// Iteration helper method to iterate from a given node in a specific direction for a specified count.
METHOD PROTECTED Iterate : POINTER TO T_List_Node
VAR_INPUT
	pStart 		: POINTER TO T_List_Node;
	Count 		: T_Capacity;
	bIterateUp 	: BOOL;
END_VAR
VAR
	i : T_Capacity;
END_VAR
Iterate := pStart;
IF Count = 0 THEN RETURN; END_IF
IF bIterateUp THEN FOR i := 0 TO Count - 1 DO Iterate := Iterate^.pNext; END_FOR RETURN; END_IF
FOR i := 0 TO Count - 1 DO Iterate := Iterate^.pPrevious; END_FOR
END_METHOD

// Adds an item to the end of the list.
METHOD Append : I_List
VAR_INPUT
	Item : ANY; // Value to store in list
END_VAR
VAR_OUTPUT
	bSuccess : BOOL;
END_VAR
Append := THIS^;

THIS^.Insert_Generic(THIS^._Count, Item, bSuccess => bSuccess);
END_METHOD

// Empties/Clears/Deletes every item in the list.
METHOD Clear : I_List
VAR
	pTmp : POINTER TO T_List_Node;
END_VAR
Clear := THIS^;

WHILE THIS^.pHead <> 0 DO
	pTmp := THIS^.pHead^.pNext;
	F_Delete_Generic(THIS^.pHead^.Data);
	__DELETE(THIS^.pHead);
	THIS^.pHead := pTmp;
	END_WHILE

THIS^._Count := 0;	
THIS^.pTail := THIS^.pLast_Accessed := 0;
THIS^.Last_Accessed_Index := -1;
THIS^.Clear_Error();
END_METHOD

// Checks if item is contained in list.
METHOD Contains : BOOL
VAR_INPUT
	Item : ANY; // Item to find in list
END_VAR
THIS^.Search(Item, bSuccess => Contains);
END_METHOD

METHOD FB_exit : BOOL
VAR_INPUT
	bInCopyCode : BOOL; // if TRUE, the exit method is called for exiting an instance that is copied afterwards (online change).
END_VAR
THIS^.Clear();
END_METHOD

// Gets item from list at specified location without removing it
METHOD Get : I_List
VAR_INPUT
	Index : T_Position; // Location of item
	Item : ANY;  // Variable to store returned item
END_VAR
VAR_OUTPUT
	bSuccess : BOOL;
END_VAR
VAR
	Tmp : T_Generic;
END_VAR
Get := THIS^;

THIS^.Get_Generic(Index, Item => Tmp, bSuccess => bSuccess);

IF NOT bSuccess THEN RETURN; END_IF

IF NOT F_Matching_Generics(Item, Tmp) THEN
	THIS^._Error_Status := F_Error(TRUE, GVL_Errors.ERR_TYPE_MISMATCH, 'Type mismatch.');
	RETURN;
	END_IF
	
F_Copy_Generic_Value(Tmp, Item);
bSuccess := TRUE;
THIS^.Clear_Error();
END_METHOD

// Returns item as a string, if type to string conversion is supported
METHOD Get_As_String : I_List
VAR_INPUT
	Index : T_Position; // Location of item
	sItem : REFERENCE TO STRING; // Variable to store returned item.
END_VAR
VAR_OUTPUT
	bSuccess : BOOL;
END_VAR
VAR
	Tmp : T_Generic;
END_VAR
Get_As_String := THIS^;

IF NOT __ISVALIDREF(sItem) THEN 
	THIS^._Error_Status := F_Error(TRUE, GVL_Errors.ERR_INVALID_REFERENCE, 'Invalid reference.');
	RETURN;
	END_IF
	
THIS^.Get_Generic(Index, Item => Tmp, bSuccess => bSuccess);

IF NOT bSuccess THEN RETURN; END_IF
	
IF NOT F_String_Convertable_Generic(Tmp) THEN 
	THIS^._Error_Status := F_Error(TRUE, GVL_Errors.ERR_NOT_SUPPORTED, 'No support for converting item at index to string.');
	RETURN;
	END_IF
	
CASE Tmp.TypeClass OF
	T_Type.TYPE_STRING:
		Tc2_Utilities.STRNCPY(ADR(sItem), Tmp.pValue, MIN(Tc2_Utilities.LEN2(ADR(sItem))+1, TO_UDINT(Tmp.diSize)));

	T_Type.TYPE_WSTRING:
		Tc2_Utilities.WSTRING_TO_STRING2(ADR(sItem), Tmp.pValue, MIN(Tc2_Utilities.LEN2(ADR(sItem))+1, TO_UDINT(Tmp.diSize)));
ELSE
	sItem := F_Generic_To_String(Tmp);
	END_CASE
	
bSuccess := TRUE;
THIS^.Clear_Error();
END_METHOD

// Gets a value from a list in it's generic form.
// (** Use carefully as this contains the pointer of the actual value in the collection. **)
// If you wish to use this it is recommeded you create a copy of the returned value using MEMMOVE or MEMCPY
METHOD Get_Generic : I_List
VAR_INPUT
	Index : T_Position; // Location of item
END_VAR
VAR_OUTPUT
	Item : T_Generic := (TypeClass := T_Type.TYPE_NONE);
	bSuccess : BOOL;
END_VAR
VAR
	pTmp : POINTER TO T_List_Node;
END_VAR
Get_Generic := THIS^;

IF Index < 0 OR_ELSE Index >= THIS^._Count THEN
	// Throw out of bounds error.
	THIS^._Error_Status := F_Error(TRUE, GVL_Errors.ERR_OUT_OF_LIMITS, 'Index out of bounds.');
	RETURN;
	END_IF
	
IF Index = 0 THEN
	Item := THIS^.pHead^.Data;
ELSIF Index = THIS^._Count - 1 THEN
	Item := THIS^.pTail^.Data;
ELSIF Index = THIS^.Last_Accessed_Index THEN
	Item := THIS^.pLast_Accessed^.Data;
ELSE
	pTmp := THIS^.Closest_Node_Iterator(Index);
	Item := pTmp^.Data;
	
	THIS^.Last_Accessed_Index := Index;
	THIS^.pLast_Accessed := pTmp;
	
	END_IF
	
bSuccess := TRUE;
THIS^.Clear_Error();
END_METHOD

// Gets the type of the item at specified location.
METHOD Get_Type_At : I_List
VAR_INPUT
	Index : T_Position;
END_VAR
VAR_OUTPUT
	Item_Type : T_Type := T_Type.TYPE_NONE;
	bSuccess : BOOL;
END_VAR
VAR
	Tmp : T_Generic;
END_VAR
Get_Type_At := THIS^;

THIS^.Get_Generic(Index, Item => Tmp, bSuccess => bSuccess);
Item_Type := Tmp.TypeClass;
END_METHOD

// Adds new item to list at specified location, if index = 0, item will be added at the front, if index = count, item will be added at the back
METHOD Insert : I_List
VAR_INPUT
	Index : T_Position; // Location of item
	Item : ANY; // Item to store in list
END_VAR
VAR_OUTPUT
	bSuccess : BOOL;
END_VAR
Insert := THIS^;

THIS^.Insert_Generic(Index, Item, bSuccess => bSuccess);
END_METHOD

// Adds new item to list at specified location using the generic form. 
// If index = 0, item will be added at the front, if index = count, item will be added at the back
METHOD Insert_Generic : I_List
VAR_INPUT
	Index 	 : T_Position; 	// Location of item
	Item 	 : T_Generic;  	// Item to store in list
END_VAR
VAR_OUTPUT
	bSuccess : BOOL;
END_VAR
VAR
	pTmp, pCurrent : POINTER TO ST_LIST_NODE;
END_VAR
Insert_Generic := THIS^;

IF Index < 0 OR_ELSE Index > THIS^._Count THEN
	// Throw out of bounds error.
	THIS^._Error_Status := F_Error(TRUE, GVL_Errors.ERR_OUT_OF_LIMITS, 'Index out of bounds.');
	RETURN;
	END_IF
	
pTmp := __NEW(ST_LIST_NODE);
pTmp^.Data := F_Clone_Generic(Item);

IF Index = 0 THEN
	//...
	pTmp^.pNext := THIS^.pHead;
	IF THIS^.pHead <> 0 THEN THIS^.pHead^.pPrevious := pTmp; END_IF
	IF THIS^.pTail = 0 THEN THIS^.pTail := pTmp; END_IF
	THIS^.pHead := pTmp;
ELSIF Index = THIS^._Count THEN
	//...
	pTmp^.pPrevious := THIS^.pTail;
	IF THIS^.pTail <> 0 THEN THIS^.pTail^.pNext := pTmp; END_IF
	THIS^.pTail := pTmp;
ELSE	
	pCurrent := THIS^.Closest_Node_Iterator(Index);
	
	pTmp^.pNext := pCurrent;
	pTmp^.pPrevious := pCurrent^.pNext;
	pCurrent^.pPrevious^.pNext := pTmp;
	pCurrent^.pPrevious := pTmp;
	
	THIS^.Last_Accessed_Index := Index;
	THIS^.pLast_Accessed := pTmp;
	END_IF
	
THIS^.Increment_Count();
bSuccess := TRUE;
THIS^.Clear_Error();
END_METHOD

// Adds an item at the front of the list.
METHOD Prepend : I_List
VAR_INPUT
	Item : ANY; // Value to store in list
END_VAR
VAR_OUTPUT
	bSuccess : BOOL;
END_VAR
Prepend := THIS^;

THIS^.Insert_Generic(0, Item, bSuccess => bSuccess);
END_METHOD

// Removes item from the list.
METHOD Remove : I_List
VAR_INPUT
	Item : ANY; // Item to remove from in list
END_VAR
VAR_OUTPUT
	bSuccess : BOOL;
END_VAR
VAR
	Tmp : T_Position;
END_VAR
Remove := THIS^;

THIS^.Search(Item, Index => Tmp, bSuccess => bSuccess);
IF NOT bSuccess THEN RETURN; END_IF 
THIS^.Remove_At(0, bSuccess => bSuccess);
END_METHOD

// Remove item at specified location 
METHOD Remove_At : I_List
VAR_INPUT
	Index : T_Position; // Location of item
END_VAR
VAR_OUTPUT
	bSuccess : BOOL;
END_VAR
VAR_INST
	pTmp, pp : POINTER TO T_List_Node;
	i : T_Position;
	MA : ARRAY[0..10] OF POINTER TO T_List_Node;
END_VAR
Remove_At := THIS^;

IF Index < 0 OR_ELSE Index >= THIS^._Count THEN
	// Throw out of bounds error.
	THIS^._Error_Status := F_Error(TRUE, GVL_Errors.ERR_OUT_OF_LIMITS, 'Index out of bounds.');
	RETURN;
	END_IF

IF Index = 0 THEN
	//...
	pTmp := THIS^.pHead;
	IF THIS^.pHead = THIS^.pTail THEN
		THIS^.pLast_Accessed := THIS^.pTail := 0;
		THIS^.Last_Accessed_Index := -1;
		END_IF
		
	THIS^.pHead := THIS^.pHead^.pNext;
	
	F_Delete_Generic(pTmp^.Data);
	__DELETE(pTmp);
	
ELSIF Index = THIS^._Count - 1 THEN
	//...
	pTmp := THIS^.pTail^.pPrevious;
	THIS^.pTail := pTmp;
	F_Delete_Generic(pTmp^.pNext^.Data);
	__DELETE(pTmp^.pNext);
ELSE
	//...	
	pTmp := THIS^.Closest_Node_Iterator(Index);
	
	// Do deletion
	pTmp^.pNext^.pPrevious := pTmp^.pPrevious;
	pTmp^.pPrevious^.pNext := pTmp^.pNext;
	
	THIS^.Last_Accessed_Index := -1;
	THIS^.pLast_Accessed := 0;
	
	THIS^.Last_Accessed_Index := Index;
	THIS^.pLast_Accessed := pTmp^.pNext;
	
	F_Delete_Generic(pTmp^.Data);
	__DELETE(pTmp);
	END_IF
	
THIS^.Decrement_Count();
bSuccess := TRUE;
THIS^.Clear_Error();
END_METHOD

// Removes item at the back of the list.
METHOD Remove_Last : I_List
VAR_OUTPUT
	bSuccess : BOOL;
END_VAR
Remove_Last := THIS^.Remove_At(THIS^._Count - 1, bSuccess => bSuccess);
END_METHOD

// Manually resize list. If list becomes smaller, item on higher locations will be deleted.
METHOD Resize : I_List
VAR_INPUT
	Size : T_Capacity; // New size of list.
END_VAR
VAR_OUTPUT
	bSuccess : BOOL;
END_VAR
VAR
	Tmp : T_Generic := (TypeClass := T_Type.TYPE_NONE);
END_VAR
Resize := THIS^;

IF Size = 0 THEN 
	THIS^.Clear();
ELSE
	WHILE THIS^._Count > Size DO THIS^.Remove_At(THIS^._Count - 1); END_WHILE
	WHILE THIS^._Count < Size DO THIS^.Insert_Generic(THIS^._Count, Tmp); END_WHILE
	END_IF
	
bSuccess := TRUE;
THIS^.Clear_Error();
END_METHOD

// Reverses the order of items in the list
METHOD Reverse : I_List
VAR_OUTPUT
	bSuccess : BOOL;
END_VAR
VAR
	pFront, pBack : POINTER TO T_List_Node;
END_VAR
Reverse := THIS^;

IF THIS^._Empty THEN RETURN; END_IF

pFront := THIS^.pHead;
pBack := THIS^.pTail;

WHILE (pFront <> pBack) AND_THEN (pFront^.pPrevious <> pBack) DO
	F_Swap_Generics(pFront^.Data, pBack^.Data);
	pFront := pFront^.pNext;
	pBack := pBack^.pPrevious;
	END_WHILE
	
bSuccess := TRUE;

THIS^.Clear_Error();
END_METHOD

// Find the location of an item in list.
METHOD Search : I_List
VAR_INPUT
	Item : ANY; // Item to find in list
END_VAR
VAR_OUTPUT
	Index : T_Position := -1; //Location of item in list 
	bSuccess : BOOL;
END_VAR
VAR
	i : T_Position;
	pTmp : POINTER TO T_List_Node;
END_VAR
Search := THIS^;

pTmp := THIS^.pHead; 
WHILE pTmp <> 0 DO
	CASE F_Compare_Generics(Item, pTmp^.Data) OF
		T_Comparison.Equal:
			bSuccess := TRUE;
			THIS^.Clear_Error();
			Index := i;
			RETURN;
		END_CASE
	pTmp := pTmp^.pNext;	
	i := i + 1;
	END_WHILE

// Throw item not found error.
THIS^._Error_Status := F_Error(TRUE, GVL_Errors.ERR_NO_OBJECT, 'Item not found.');
END_METHOD

// Changes the item at the specified location in the list.
METHOD Set : I_List
VAR_INPUT
	Index 	: T_Position; // Location of item
	Item 	: ANY; 	// Item to store in list
END_VAR
VAR_OUTPUT
	bSuccess : BOOL;
END_VAR
Set := THIS^;

THIS^.Set_Generic(Index, Item, bSuccess => bSuccess);
END_METHOD

// Changes the item at the specified location in the list in it's generic form.
METHOD Set_Generic : I_List
VAR_INPUT
	Index : T_Position; // Location of item
	Item : T_Generic; // Item to store in list
END_VAR
VAR_OUTPUT
	bSuccess : BOOL;
END_VAR
VAR
	pTmp : POINTER TO T_List_Node;
END_VAR
Set_Generic := THIS^;

IF Index < 0 OR_ELSE Index >= THIS^._Count THEN
	// Throw out of bounds error.
	THIS^._Error_Status := F_Error(TRUE, GVL_Errors.ERR_OUT_OF_LIMITS, 'Index out of bounds.');
	RETURN;
	END_IF
	
IF Index = 0 THEN
	F_Delete_Generic(THIS^.pHead^.Data);
	THIS^.pHead^.Data := F_Clone_Generic(Item);
ELSIF Index = THIS^._Count - 1 THEN
	F_Delete_Generic(THIS^.pTail^.Data);
	THIS^.pTail^.Data := F_Clone_Generic(Item);
ELSIF Index = THIS^.Last_Accessed_Index THEN
	F_Delete_Generic(THIS^.pLast_Accessed^.Data);
	THIS^.pLast_Accessed^.Data := F_Clone_Generic(Item);
ELSE
	pTmp := THIS^.Closest_Node_Iterator(Index);
	F_Delete_Generic(pTmp^.Data);
	pTmp^.Data := F_Clone_Generic(Item);

	THIS^.Last_Accessed_Index := Index;
	THIS^.pLast_Accessed := pTmp;
	END_IF
	
bSuccess := TRUE;
THIS^.Clear_Error();
END_METHOD

// Swaps item at index A with item at index B.
METHOD Swap : I_List
VAR_INPUT
	Index_A, Index_B : T_Position;
END_VAR
VAR_OUTPUT
	bSuccess : BOOL;
END_VAR
Swap := THIS^;

IF Index_A < 0 OR_ELSE Index_A >= THIS^._Count OR_ELSE Index_B < 0 OR_ELSE Index_B >= THIS^._Count THEN
	THIS^._Error_Status := F_Error(TRUE, GVL_Errors.ERR_OUT_OF_LIMITS, 'Index out of bounds.');
	RETURN;
	END_IF
	
bSuccess := F_Swap_Generics(THIS^.Closest_Node_Iterator(Index_A)^.Data, THIS^.Closest_Node_Iterator(Index_B)^.Data);
THIS^.Clear_Error();
END_METHOD

END_FUNCTION_BLOCK

// POUs/Function Blocks/Collections/FB_Hash_Map
// A collection of key value pairs items.
{attribute 'enable_dynamic_creation'}
{attribute 'no_assign'}
{attribute 'no_explicit_call' := 'direct call for this function block is not allowed'}
FUNCTION_BLOCK FB_Hash_Map EXTENDS FB_Collection
VAR
END_VAR

END_FUNCTION_BLOCK

// POUs/Function Blocks/Collections/FB_Hash_Set
// A collection that contains no duplicate items.
{attribute 'enable_dynamic_creation'}
{attribute 'no_assign'}
{attribute 'no_explicit_call' := 'direct call for this function block is not allowed'}
FUNCTION_BLOCK FB_Hash_Set EXTENDS FB_Collection
VAR
END_VAR

END_FUNCTION_BLOCK

// POUs/Function Blocks/Collections/FB_Queue
// A collection whose access/mutation of items is first-in, first-out.
{attribute 'enable_dynamic_creation'}
{attribute 'no_assign'}
{attribute 'no_explicit_call' := 'direct call for this function block is not allowed'}
FUNCTION_BLOCK FINAL FB_Queue EXTENDS FB_Collection IMPLEMENTS I_Queue//, I_Enumerable, I_Copyable
VAR
	fbList : FB_List := ();
END_VAR

// Gets an immutable list of the items in the queue.
PROPERTY _Values : I_Immutable_List
GET
VAR_INST
	fbImmutable_List : FB_Immutable_List := (ipList := THIS^.fbList);
END_VAR
_Values := fbImmutable_List;
END_GET
END_PROPERTY

// Empties/Clears/Deletes every item in the queue.
METHOD Clear : I_Queue
Clear := THIS^;

THIS^.fbList.Clear();

THIS^._Error_Status :=  THIS^.fbList._Error_Status;
THIS^._Count := THIS^.fbList._Count;
END_METHOD

// Removes item at the front the queue.
METHOD Dequeue : I_Queue
VAR_OUTPUT
	bSuccess : BOOL;
END_VAR
Dequeue := THIS^;

THIS^.fbList.Remove_At(0, bSuccess => bSuccess);

THIS^._Error_Status := THIS^.fbList._Error_Status;
THIS^._Count := THIS^.fbList._Count;
END_METHOD

// Adds item at the back of the queue.
METHOD Enqueue : I_Queue
VAR_INPUT
	Item : ANY; // Variable containg data to store on the queue.
END_VAR
VAR_OUTPUT
	bSuccess : BOOL;
END_VAR
Enqueue := THIS^;

THIS^.fbList.Insert_Generic(THIS^.fbList._Count, Item, bSuccess => bSuccess);

THIS^._Error_Status :=  THIS^.fbList._Error_Status;
THIS^._Count := THIS^.fbList._Count;
END_METHOD

// Adds item at the front of the queue.
METHOD Enqueue_At_Front : I_Queue
VAR_INPUT
	Item : ANY; // Variable containg data to store on the queue.
END_VAR
VAR_OUTPUT
	bSuccess : BOOL;
END_VAR
Enqueue_At_Front := THIS^;

THIS^.fbList.Insert_Generic(0, Item, bSuccess => bSuccess);

THIS^._Error_Status :=  THIS^.fbList._Error_Status;
THIS^._Count := THIS^.fbList._Count;
END_METHOD

// Adds a generic item at the back of the queue.
METHOD Enqueue_Generic : I_Queue
VAR_INPUT
	Item : T_Generic; // Item to store.
	bAt_Front : BOOL; // Enqueues at front if set to TRUE.
END_VAR
VAR_OUTPUT
	bSuccess : BOOL;
END_VAR
Enqueue_Generic := THIS^;

IF bAt_Front THEN
	THIS^.fbList.Insert_Generic(0, Item, bSuccess => bSuccess);
ELSE
	THIS^.fbList.Insert_Generic(THIS^.fbList._Count, Item, bSuccess => bSuccess);
	END_IF
	
THIS^._Error_Status :=  THIS^.fbList._Error_Status;
THIS^._Count := THIS^.fbList._Count;
END_METHOD

// Gets the item at the front of the queue.
METHOD Get : I_Queue
VAR_INPUT
	Item : ANY; // Variable to store returned item value
END_VAR
VAR_OUTPUT
	bSuccess : BOOL;
END_VAR
Get := THIS^;

THIS^.fbList.Get(0, Item, bSuccess => bSuccess);

THIS^._Error_Status := THIS^.fbList._Error_Status;
END_METHOD

// Gets the item at the front of the queue as a generic.
METHOD Get_Generic : I_Queue
VAR_OUTPUT
	Item : T_Generic; // Variable to store returned item value
	bSuccess : BOOL;
END_VAR
Get_Generic := THIS^;

THIS^.fbList.Get_Generic(0, Item => Item, bSuccess => bSuccess);

THIS^._Error_Status := THIS^.fbList._Error_Status;
END_METHOD

// Reverses the order of the items in the queue.
METHOD Reverse : I_Queue
VAR_OUTPUT
	bSuccess : BOOL;
END_VAR
Reverse := THIS^;

THIS^.fbList.Reverse(bSuccess => bSuccess);

THIS^._Error_Status :=  THIS^.fbList._Error_Status;
END_METHOD

END_FUNCTION_BLOCK

// POUs/Function Blocks/Collections/FB_Stack
// A collection whose access/mutation of items is last-in, first-out.
{attribute 'enable_dynamic_creation'}
{attribute 'no_assign'}
{attribute 'no_explicit_call' := 'direct call for this function block is not allowed'}
FUNCTION_BLOCK FINAL FB_Stack EXTENDS FB_Collection IMPLEMENTS I_Stack //, I_Enumerable, I_Copyable
VAR
	fbList : FB_List;
END_VAR

// Gets an immutable list of the items in the stack.
PROPERTY _Values : I_Immutable_List
GET
VAR_INST
	fbImmutable_List : FB_Immutable_List := (ipList := THIS^.fbList);
END_VAR
_Values := fbImmutable_List;
END_GET
END_PROPERTY

// Empties/Clears/Deletes every item in the stack.
METHOD Clear : I_Stack
Clear := THIS^;

THIS^.fbList.Clear();

THIS^._Error_Status :=  THIS^.fbList._Error_Status;
THIS^._Count := THIS^.fbList._Count;
END_METHOD

// Gets item at the top of the stack.
METHOD Get : I_Stack
VAR_INPUT
	Item : ANY; // Variable to store returned item value. 
END_VAR
VAR_OUTPUT
	bSuccess : BOOL;
END_VAR
Get := THIS^;

THIS^.fbList.Get(0, Item, bSuccess => bSuccess);

THIS^._Error_Status := THIS^.fbList._Error_Status;
END_METHOD

// Gets item at the top of the stack as a generic.
METHOD Get_Generic : I_Stack
VAR_OUTPUT
	Item : T_Generic; // Variable to store returned item value
	bSuccess : BOOL;
END_VAR
Get_Generic := THIS^;

THIS^.fbList.Get_Generic(0, Item => Item, bSuccess => bSuccess);

THIS^._Error_Status := THIS^.fbList._Error_Status;
END_METHOD

// Removes item at the top of the stack without returning anything.
METHOD Pop : I_Stack
VAR_OUTPUT
	bSuccess : BOOL;
END_VAR
Pop := THIS^;

THIS^.fbList.Remove_At(0, bSuccess => bSuccess);

THIS^._Error_Status := THIS^.fbList._Error_Status;
THIS^._Count := THIS^.fbList._Count;
END_METHOD

// Add item to the top of the stack.
METHOD Push : I_Stack
VAR_INPUT
	Item : ANY; // Item to store.
END_VAR
VAR_OUTPUT
	bSuccess : BOOL;
END_VAR
Push := THIS^;

THIS^.fbList.Insert_Generic(0, Item, bSuccess => bSuccess);

THIS^._Error_Status :=  THIS^.fbList._Error_Status;
THIS^._Count := THIS^.fbList._Count;
END_METHOD

// Add generic item to the top of the stack.
METHOD Push_Generic : I_Stack
VAR_INPUT
	Item : T_Generic; // Item to store.
END_VAR
VAR_OUTPUT
	bSuccess : BOOL;
END_VAR
Push_Generic := THIS^;

THIS^.fbList.Insert_Generic(0, Item, bSuccess => bSuccess);

THIS^._Error_Status :=  THIS^.fbList._Error_Status;
THIS^._Count := THIS^.fbList._Count;
END_METHOD

// Reverses order of items on stack.
METHOD Reverse : I_Stack
VAR_OUTPUT
	bSuccess : BOOL;
END_VAR
Reverse := THIS^;

THIS^.fbList.Reverse(bSuccess => bSuccess);

THIS^._Error_Status :=  THIS^.fbList._Error_Status;
END_METHOD

END_FUNCTION_BLOCK

// POUs/Function Blocks/Collections/FB_Tree_Map
// A collection of key-value pair items implemented using an iterative AVL Tree. 
// Keys and values can be retrieved as an immutable list (whose base is FB_ArrayList) via 4 traversal methods; Inorder, Preorder, Postorder and Level Order.
// This data structure was implemented with the help of Max Goren's iterative AVL tree in C++. See Function Block's body for more details.
{attribute 'enable_dynamic_creation'}
{attribute 'no_assign'}
{attribute 'no_explicit_call' := 'direct call for this function block is not allowed'}
FUNCTION_BLOCK FB_Tree_Map EXTENDS FB_Collection IMPLEMENTS I_Tree_Map //, I_Enumerable, I_Copyable
VAR
	pRoot : POINTER TO T_AVL_Map_Node;
	Traversal : T_BST_Traversal := T_BST_Traversal.In_Order; 
	pKeys, pValues : POINTER TO FB_Array_List;
END_VAR

(*
	https://github.com/maxgoren
	https://github.com/maxgoren/Algorithms/
	http://www.maxgcoding.com/iterative-avl-trees-insertion/
	http://www.maxgcoding.com/iterative-avl-trees-deletion/

	MIT License
	
	Copyright (c) 2021 Max Goren
	
	Permission is hereby granted, free of charge, to any person obtaining a copy
	of this software and associated documentation files (the "Software"), to deal
	in the Software without restriction, including without limitation the rights
	to use, copy, modify, merge, publish, distribute, sublicense, and/or sell
	copies of the Software, and to permit persons to whom the Software is
	furnished to do so, subject to the following conditions:
	
	The above copyright notice and this permission notice shall be included in all
	copies or substantial portions of the Software.
	
	THE SOFTWARE IS PROVIDED "AS IS", WITHOUT WARRANTY OF ANY KIND, EXPRESS OR
	IMPLIED, INCLUDING BUT NOT LIMITED TO THE WARRANTIES OF MERCHANTABILITY,
	FITNESS FOR A PARTICULAR PURPOSE AND NONINFRINGEMENT. IN NO EVENT SHALL THE
	AUTHORS OR COPYRIGHT HOLDERS BE LIABLE FOR ANY CLAIM, DAMAGES OR OTHER
	LIABILITY, WHETHER IN AN ACTION OF CONTRACT, TORT OR OTHERWISE, ARISING FROM,
	OUT OF OR IN CONNECTION WITH THE SOFTWARE OR THE USE OR OTHER DEALINGS IN THE
	SOFTWARE.
*)

// Performs rotation and updates heights until tree is balanced.
METHOD PROTECTED Balance
VAR_INPUT
    pNode : POINTER TO T_AVL_Map_Node;
END_VAR
VAR 
	pTmp : POINTER TO T_AVL_Map_Node;
    Balance_Factor : T_Position;
END_VAR
WHILE pNode <> 0 AND_THEN pNode^.pParent <> 0 DO
	pTmp := pNode^.pParent;
	
	THIS^.Update_Height(pTmp);
	
	IF THIS^.Get_Balance(pTmp) < -1 THEN
		IF THIS^.Get_Balance(pTmp^.pRight) > 0 THEN THIS^.Rotate_Right(pTmp^.pRight); END_IF
		THIS^.Rotate_Left(pTmp);
		
	ELSIF THIS^.Get_Balance(pTmp) > 1 THEN
		IF THIS^.Get_Balance(pTmp^.pLeft) < 0 THEN THIS^.Rotate_Left(pTmp^.pLeft); END_IF
		THIS^.Rotate_Right(pTmp);
		END_IF
	
	pNode := pNode^.pParent;
	END_WHILE
END_METHOD

// Deletes the node and its tree/sub-trees.
{warning disable C0394}
METHOD PROTECTED Clear_Node
VAR_INPUT
	pRoot : POINTER TO T_AVL_Map_Node;
END_VAR
VAR
	fbNode_Stack : FB_Stack;
	pTmp : POINTER TO T_AVL_Map_Node;
END_VAR
IF pRoot = 0 THEN RETURN; END_IF

fbNode_Stack.Push(pRoot);

WHILE NOT fbNode_Stack._Empty DO
	fbNode_Stack.Get(pTmp);
	fbNode_Stack.Pop();
	
	IF pTmp^.pRight <> 0 THEN fbNode_Stack.Push(pTmp^.pRight); END_IF
	IF pTmp^.pLeft <> 0 THEN fbNode_Stack.Push(pTmp^.pLeft); END_IF
	
	THIS^.Delete_Node(pTmp);
	END_WHILE
END_METHOD

// Creates a new node in dynamic memory with a clone of the generic item as it data.
METHOD PROTECTED Create_Node : POINTER TO ST_AVL_MAP_NODE
VAR_INPUT
	Key, Value : T_Generic;
END_VAR
Create_Node := __NEW(ST_AVL_MAP_NODE);
Create_Node^.Key := F_Clone_Generic(Key);
Create_Node^.Value := F_Clone_Generic(Value);
END_METHOD

// Safety deletes node.
// If the node and/or it's value/data is in dynamic memory it/they will be deleted.
METHOD PROTECTED Delete_Node
VAR_INPUT
	pNode : REFERENCE TO POINTER TO T_AVL_Map_Node;
END_VAR
IF (pNode = 0) THEN RETURN; END_IF 

F_Delete_Generic(pNode^.Key);
F_Delete_Generic(pNode^.Value);

CASE Tc2_System.F_CheckMemoryArea(pNode, 1) OF
	Tc2_System.E_TcMemoryArea.Dynamic: __DELETE(pNode);
ELSE
	pNode := 0;
	END_CASE
END_METHOD

// Finds the node with the smallest item in a tree or sub-tree.
METHOD PROTECTED Find_Minimum_Node : POINTER TO T_AVL_Node
VAR_INPUT
	pNode : POINTER TO T_AVL_Map_Node;
END_VAR
IF pNode = 0 THEN RETURN; END_IF

WHILE pNode^.pLeft <> 0 DO
	pNode := pNode^.pLeft;
	END_WHILE
	
Find_Minimum_Node := pNode;
END_METHOD

// Gets the difference between the left and right sub-trees.
METHOD PROTECTED Get_Balance : T_Position
VAR_INPUT
	pNode : POINTER TO T_AVL_Map_Node;
END_VAR
Get_Balance :=  THIS^.Get_Height(pNode^.pLeft) - THIS^.Get_Height(pNode^.pRight);
END_METHOD

// Safely gets the height of a sub-tree.
METHOD PROTECTED Get_Height : T_Position
VAR_INPUT
	pNode : POINTER TO T_AVL_Map_Node;
END_VAR
Get_Height := SEL(pNode <> 0, -1, pNode^.Height);
END_METHOD

// Moves from node at source into the position of the destination.
METHOD PROTECTED Move_Node
VAR_INPUT
	pDestination, pSource : POINTER TO T_AVL_Map_Node;
END_VAR
IF pDestination^.pParent = 0 THEN
	THIS^.pRoot := pSource;
ELSIF pDestination = pDestination^.pParent^.pLeft THEN
	pDestination^.pParent^.pLeft := pSource;
ELSE
	pDestination^.pParent^.pRight := pSource;
	END_IF
	
IF pSource <> 0 THEN
	pSource^.pParent := pDestination^.pParent;
	END_IF
END_METHOD

// Finds and removes a node from a tree/sub-tree.
METHOD PROTECTED Remove_Node
VAR_INPUT
	pNode : POINTER TO T_AVL_Map_Node;
END_VAR
VAR
	pTmp, pSuccessor : POINTER TO T_AVL_Map_Node;
END_VAR
pTmp := pNode;

IF pNode^.pLeft = 0 THEN
	THIS^.Move_Node(pNode, pNode^.pRight);
ELSIF pNode^.pRight = 0 THEN 
	THIS^.Move_Node(pNode, pNode^.pLeft);
ELSE
	pSuccessor := THIS^.Find_Minimum_Node(pNode^.pRight);
	IF pSuccessor^.pParent <> pNode THEN 
		THIS^.Move_Node(pSuccessor, pSuccessor^.pRight);
		pSuccessor^.pRight := pNode^.pRight;
		pSuccessor^.pRight^.pParent := pSuccessor;
		END_IF
	THIS^.Move_Node(pNode, pSuccessor);
	pSuccessor^.pLeft := pNode^.pLeft;
	pSuccessor^.pLeft^.pParent := pSuccessor;
	END_IF

THIS^.Delete_Node(pTmp);
END_METHOD

// Rotates a tree/sub-tree left.
METHOD PROTECTED Rotate_Left
VAR_INPUT
    pX : POINTER TO T_AVL_Map_Node;
END_VAR
VAR
    pY : POINTER TO T_AVL_Map_Node := pX^.pRight;
END_VAR
IF pY <> 0 THEN
	pX^.pRight := pY^.pLeft;
	IF pY^.pLeft <> 0 THEN pY^.pLeft^.pParent := pX; END_IF
	pY^.pParent := pX^.pParent;
	END_IF
	
IF pX^.pParent = 0 THEN
	THIS^.pRoot := pY;
ELSIF pX = pX^.pParent^.pLeft THEN
	pX^.pParent^.pLeft := pY;
ELSE
	pX^.pParent^.pRight := pY;
	END_IF
	
IF pY <> 0 THEN pY^.pLeft := pX; END_IF
	
pX^.pParent := pY;
THIS^.Update_Height(pX);
THIS^.Update_Height(pY);
END_METHOD

// Rotates a tree/sub-tree right.
METHOD PROTECTED Rotate_Right
VAR_INPUT
    pX : POINTER TO T_AVL_Map_Node;
END_VAR
VAR
    pY : POINTER TO T_AVL_Map_Node := pX^.pLeft;
END_VAR
IF pY <> 0 THEN
	pX^.pLeft := pY^.pRight;
	IF pY^.pRight <> 0 THEN pY^.pRight^.pParent := pX; END_IF
	pY^.pParent := pX^.pParent;
	END_IF
	
IF pX^.pParent = 0 THEN
	THIS^.pRoot := pY;
ELSIF pX = pX^.pParent^.pLeft THEN
	pX^.pParent^.pLeft := pY;
ELSE
	pX^.pParent^.pRight := pY;
	END_IF
	
IF pY <> 0 THEN pY^.pRight := pX; END_IF
	
pX^.pParent := pY;
THIS^.Update_Height(pX);
THIS^.Update_Height(pY);
END_METHOD

// Checks if an item is in a tree/ sub-tree.
METHOD PROTECTED Search_Node : POINTER TO T_AVL_Map_Node
VAR_INPUT
	pNode : POINTER TO T_AVL_Map_Node;
	Key : T_Generic;
END_VAR
WHILE pNode <> 0 DO
	CASE F_Compare_Generics(Key, pNode^.Key) OF
		T_Comparison.Less	: pNode := pNode^.pLeft;
		T_Comparison.Greater: pNode := pNode^.pRight; 
		T_Comparison.Equal	: 
			Search_Node := pNode;
			RETURN;
		END_CASE
	END_WHILE
END_METHOD

METHOD PROTECTED Update_Height
VAR_INPUT
	pNode : POINTER TO T_AVL_Map_Node;
END_VAR
pNode^.Height := 1 + MAX(THIS^.Get_Height(pNode^.pLeft), THIS^.Get_Height(pNode^.pRight));
END_METHOD

// Traversal method for retrieving keys and values in the tree map set.
PROPERTY _Traversal : T_BST_Traversal
GET
_Traversal := THIS^.Traversal;
END_GET
SET
THIS^.Traversal := _Traversal;
END_SET
END_PROPERTY

// Empties/Clears/Deletes every item in the map.
METHOD Clear : I_Map
Clear := THIS^;

THIS^.Clear_Node(THIS^.pRoot);

IF THIS^.pKeys <> 0 THEN  __DELETE(THIS^.pKeys); END_IF
IF THIS^.pValues <> 0 THEN  __DELETE(THIS^.pValues); END_IF

THIS^.pRoot := 0;
THIS^._Count := 0;
END_METHOD

// Checks if key is contained in the map.
METHOD Contains : BOOL
VAR_INPUT
	Key : ANY; // Key to find.
END_VAR
Contains := THIS^.Search_Node(THIS^.pRoot, Key) <> 0;
END_METHOD

{attribute 'hide'}
METHOD FB_exit : BOOL
VAR_INPUT
	bInCopyCode : BOOL; // if TRUE, the exit method is called for exiting an instance that is copied afterwards (online change).
END_VAR
// If this is an online change or this collection is empty then ignore. 
IF bInCopyCode THEN RETURN; END_IF

THIS^.Clear();
END_METHOD

// Gets the value associated with the specified key without removing it from the map.
METHOD Get : I_Map
VAR_INPUT
	Key : ANY; // Key used to identify stored value
	Value : ANY; // Variable to store requested data 
END_VAR
VAR_OUTPUT
	bSuccess : BOOL;
END_VAR
VAR
	Tmp : T_Generic;
END_VAR
Get := THIS^;

THIS^.Get_Generic(Key, Value => Tmp, bSuccess => bSuccess);

IF NOT bSuccess THEN RETURN; END_IF

IF NOT F_Matching_Generics(Value, Tmp) THEN
	THIS^._Error_Status := F_Error(TRUE, GVL_Errors.ERR_TYPE_MISMATCH, 'Type mismatch.');
	RETURN;
	END_IF
	
F_Copy_Generic_Value(Tmp, Value);
bSuccess := TRUE;
THIS^.Clear_Error();
END_METHOD

// Returns value as a string, if type to string conversion is supported.
METHOD Get_As_String : I_Map
VAR_INPUT
	Key : ANY; // Key used to identify stored value
	sValue : REFERENCE TO STRING; // Variable to store returned item.
END_VAR
VAR_OUTPUT
	bSuccess : BOOL;
END_VAR
VAR
	Tmp : T_Generic;
END_VAR
Get_As_String := THIS^;

IF NOT __ISVALIDREF(sValue) THEN 
	THIS^._Error_Status := F_Error(TRUE, GVL_Errors.ERR_INVALID_REFERENCE, 'Invalid reference.');
	RETURN;
	END_IF
	
THIS^.Get_Generic(Key, Value => Tmp, bSuccess => bSuccess);

IF NOT bSuccess THEN RETURN; END_IF

IF NOT F_String_Convertable_Generic(Tmp) THEN 
	THIS^._Error_Status := F_Error(TRUE, GVL_Errors.ERR_NOT_SUPPORTED, 'No support for converting item at index to string.');
	RETURN;
	END_IF
	
CASE Tmp.TypeClass OF
	T_Type.TYPE_STRING:
		Tc2_Utilities.STRNCPY(ADR(sValue), Tmp.pValue, MIN(Tc2_Utilities.LEN2(ADR(sValue))+1, TO_UDINT(Tmp.diSize)));

	T_Type.TYPE_WSTRING:
		Tc2_Utilities.WSTRING_TO_STRING2(ADR(sValue), Tmp.pValue, MIN(Tc2_Utilities.LEN2(ADR(sValue))+1, TO_UDINT(Tmp.diSize)));
ELSE
	sValue := F_Generic_To_String(Tmp);
	END_CASE
	
bSuccess := TRUE;
THIS^.Clear_Error();
END_METHOD

// Gets the value in its generic form associated with the specified key in its generic form without removing it from the map.
// (** Use carefully as this contains the pointer of the actual value in the collection. **)
// If you wish to use this it is recommeded you create a copy of the returned value using MEMMOVE or MEMCPY
METHOD Get_Generic : I_Map
VAR_INPUT
	Key : T_Generic; // Key used to identify stored value
END_VAR
VAR_OUTPUT
	Value : T_Generic := (TypeClass := T_Type.TYPE_NONE); // Variable to store requested data 
	bSuccess : BOOL;
END_VAR
VAR
	pTmp : POINTER TO T_AVL_Map_Node;
END_VAR
Get_Generic := THIS^;

pTmp := THIS^.Search_Node(THIS^.pRoot, Key);
bSuccess := pTmp <> 0;

IF bSuccess THEN RETURN; END_IF

Value := pTmp^.Value;
THIS^.Clear_Error();
END_METHOD

// Gets an immutable list of the keys.
{warning disable C0394}
METHOD Get_Keys : I_Immutable_List
VAR_INST
	fbImmutable_List : FB_Immutable_List;
END_VAR
VAR
	pCurrent : POINTER TO T_AVL_Map_Node;
	fbNode_Buffer : FB_Queue;
END_VAR
IF THIS^.pKeys = 0 THEN THIS^.pKeys := __NEW(FB_Array_List(Initial_Capacity := 0)); END_IF
fbImmutable_List(ipList := THIS^.pKeys^);
Get_Keys := fbImmutable_List;

THIS^.pKeys^.Clear();

IF THIS^.pRoot = 0 THEN RETURN; END_IF

fbNode_Buffer.Enqueue(THIS^.pRoot);

WHILE NOT fbNode_Buffer._Empty DO
	fbNode_Buffer.Get(pCurrent).Dequeue();
	
	CASE THIS^._Traversal OF
		T_BST_Traversal.In_Order:
			IF pCurrent^.pLeft <> 0 THEN fbNode_Buffer.Enqueue_At_Front(pCurrent^.pLeft); END_IF
			THIS^.pKeys^.Insert_Generic(THIS^.pKeys^._Count, pCurrent^.Value);
			IF pCurrent^.pRight <> 0 THEN fbNode_Buffer.Enqueue_At_Front(pCurrent^.pRight); END_IF
			
		T_BST_Traversal.Pre_Order:
			THIS^.pKeys^.Insert_Generic(THIS^.pKeys^._Count, pCurrent^.Value);
			IF pCurrent^.pLeft <> 0 THEN fbNode_Buffer.Enqueue_At_Front(pCurrent^.pLeft); END_IF
			IF pCurrent^.pRight <> 0 THEN fbNode_Buffer.Enqueue_At_Front(pCurrent^.pRight); END_IF
			
		T_BST_Traversal.Post_Order:
			IF pCurrent^.pLeft <> 0 THEN fbNode_Buffer.Enqueue_At_Front(pCurrent^.pLeft); END_IF
			IF pCurrent^.pRight <> 0 THEN fbNode_Buffer.Enqueue_At_Front(pCurrent^.pRight); END_IF
			THIS^.pKeys^.Insert_Generic(THIS^.pKeys^._Count, pCurrent^.Value);
			
		T_BST_Traversal.Level_Order:
			THIS^.pKeys^.Insert_Generic(THIS^.pKeys^._Count, pCurrent^.Value);
			IF pCurrent^.pLeft <> 0 THEN fbNode_Buffer.Enqueue(pCurrent^.pLeft); END_IF
			IF pCurrent^.pRight <> 0 THEN fbNode_Buffer.Enqueue(pCurrent^.pRight); END_IF
	ELSE
		RETURN;
		END_CASE
	END_WHILE
END_METHOD

// Gets an immutable list of the values.
{warning disable C0394}
METHOD Get_Values : I_Immutable_List
VAR_INST
	fbImmutable_List : FB_Immutable_List;
END_VAR
VAR
	pCurrent : POINTER TO T_AVL_Map_Node;
	fbNode_Buffer : FB_Queue;
END_VAR
IF THIS^.pValues = 0 THEN THIS^.pValues := __NEW(FB_Array_List(Initial_Capacity := 0)); END_IF
fbImmutable_List(ipList := THIS^.pValues^);
Get_Values := fbImmutable_List;

THIS^.pValues^.Clear();

IF THIS^.pRoot = 0 THEN RETURN; END_IF

fbNode_Buffer.Enqueue(THIS^.pRoot);

WHILE NOT fbNode_Buffer._Empty DO
	fbNode_Buffer.Get(pCurrent).Dequeue();
	
	CASE THIS^._Traversal OF
		T_BST_Traversal.In_Order:
			IF pCurrent^.pLeft <> 0 THEN fbNode_Buffer.Enqueue_At_Front(pCurrent^.pLeft); END_IF
			THIS^.pValues^.Insert_Generic(THIS^.pValues^._Count, pCurrent^.Value);
			IF pCurrent^.pRight <> 0 THEN fbNode_Buffer.Enqueue_At_Front(pCurrent^.pRight); END_IF
			
		T_BST_Traversal.Pre_Order:
			THIS^.pValues^.Insert_Generic(THIS^.pValues^._Count, pCurrent^.Value);
			IF pCurrent^.pLeft <> 0 THEN fbNode_Buffer.Enqueue_At_Front(pCurrent^.pLeft); END_IF
			IF pCurrent^.pRight <> 0 THEN fbNode_Buffer.Enqueue_At_Front(pCurrent^.pRight); END_IF
			
		T_BST_Traversal.Post_Order:
			IF pCurrent^.pLeft <> 0 THEN fbNode_Buffer.Enqueue_At_Front(pCurrent^.pLeft); END_IF
			IF pCurrent^.pRight <> 0 THEN fbNode_Buffer.Enqueue_At_Front(pCurrent^.pRight); END_IF
			THIS^.pValues^.Insert_Generic(THIS^.pValues^._Count, pCurrent^.Value);
			
		T_BST_Traversal.Level_Order:
			THIS^.pValues^.Insert_Generic(THIS^.pValues^._Count, pCurrent^.Value);
			IF pCurrent^.pLeft <> 0 THEN fbNode_Buffer.Enqueue(pCurrent^.pLeft); END_IF
			IF pCurrent^.pRight <> 0 THEN fbNode_Buffer.Enqueue(pCurrent^.pRight); END_IF
	ELSE
		RETURN;
		END_CASE
	END_WHILE
END_METHOD

// Insert an element with the provided key and value to the map.
METHOD Insert : I_Map
VAR_INPUT
	Key : ANY; // Key used to identify stored value
	Value : ANY; // Value to store in map with key
END_VAR
VAR_OUTPUT
	bSuccess : BOOL;
END_VAR
Insert := THIS^.Insert_Generic(Key, Value, FALSE, bSuccess => bSuccess);
END_METHOD

// Insert an element with the provided key and value in their generic forms to the map.
METHOD Insert_Generic : I_Map
VAR_INPUT
	Key : T_Generic; // Key used to identify stored value
	Value : T_Generic; // Value to store in map with key
	bUpdate : BOOL; // If this is true the value will be updated if the key already exists.
END_VAR
VAR_OUTPUT
	bSuccess : BOOL;
END_VAR
VAR
	pCurrent, pPrevious : POINTER TO T_AVL_Map_Node;
END_VAR
Insert_Generic := THIS^;

pCurrent := THIS^.pRoot;
pPrevious := pCurrent;

WHILE pCurrent <> 0 DO
	pPrevious := pCurrent;
	CASE F_Compare_Generics(Key, pCurrent^.Key) OF
		T_Comparison.Less 	 : pCurrent := pCurrent^.pLeft;
		T_Comparison.Greater : pCurrent := pCurrent^.pRight;
		T_Comparison.Equal 	 : 
			IF bUpdate THEN
				F_Delete_Generic(pCurrent^.Value);
				pCurrent^.Value := F_Clone_Generic(Value);
				bSuccess := TRUE;
				THIS^.Clear_Error();
			ELSE
				THIS^._Error_Status := F_Error(TRUE, GVL_Errors.ERR_DUPLICATE, 'Duplicate key.');
				END_IF
			RETURN;
	ELSE
		THIS^._Error_Status := F_Error(TRUE, GVL_Errors.ERR_NOT_SUPPORTED, 'Invalid comparison.');
		RETURN;
		END_CASE
	END_WHILE
	
pCurrent := THIS^.Create_Node(Key, Value);

IF pPrevious = 0 THEN
	THIS^.pRoot := pCurrent;
ELSE
	CASE F_Compare_Generics(Key, pPrevious^.Key) OF
		T_Comparison.Less: pPrevious^.pLeft := pCurrent;
	ELSE
		pPrevious^.pRight := pCurrent;
		END_CASE
	END_IF
	
pCurrent^.pParent := pPrevious;
	
THIS^.Balance(pCurrent);

bSuccess := TRUE;
THIS^.Increment_Count();
THIS^.Clear_Error();
END_METHOD

// Removes value with the specified key from the map.
METHOD Remove : I_Map
VAR_INPUT
	Key : ANY; // Key used to identify stored value
END_VAR
VAR_OUTPUT
	bSuccess : BOOL;
END_VAR
Remove := THIS^.Remove_Generic(Key, bSuccess => bSuccess);
END_METHOD

// Removes value with the specified key in its generic form from the map.
METHOD Remove_Generic : I_Map
VAR_INPUT
	Key : T_Generic; // Key used to identify stored value
END_VAR
VAR_OUTPUT
	bSuccess : BOOL;
END_VAR
VAR
	pTmp : POINTER TO T_AVL_Map_Node;
END_VAR
Remove_Generic := THIS^;

pTmp := THIS^.Search_Node(THIS^.pRoot, Key);

bSuccess := pTmp <> 0;

IF NOT bSuccess THEN
	THIS^._Error_Status := F_Error(TRUE, GVL_Errors.ERR_NO_OBJECT, 'Key not found.');
	RETURN;
	END_IF

THIS^.Remove_Node(pTmp);
THIS^.Balance(pTmp);

THIS^.Decrement_Count();
THIS^.Clear_Error();

IF THIS^._Empty THEN THIS^.pRoot := 0; END_IF
END_METHOD

// Updates the value an element with the provided key and value in the map.
METHOD Update : I_Map
VAR_INPUT
	Key 	: ANY; // Key used to identify stored value
	Value 	: ANY; // Value to store in map with key
END_VAR
VAR_OUTPUT
	bSuccess : BOOL;
END_VAR
VAR
	pTmp : POINTER TO T_AVL_Map_Node;
END_VAR
Update := THIS^;

pTmp := THIS^.Search_Node(THIS^.pRoot, Key);

bSuccess := pTmp <> 0;

IF NOT bSuccess THEN 
	THIS^._Error_Status := F_Error(TRUE, GVL_Errors.ERR_NO_OBJECT, 'Key not found.');
	RETURN;
	END_IF
	
F_Delete_Generic(pTmp^.Value);
pTmp^.Value := F_Clone_Generic(Value);
THIS^.Clear_Error();
END_METHOD

// Updates a value in the map for a given key. If the key doesnt exist, it will be inserted.
METHOD Upsert : I_Map
VAR_INPUT
	Key 	: ANY; // Key used to identify stored value
	Value 	: ANY; // Value to store in map with key
END_VAR
VAR_OUTPUT
	bSuccess : BOOL;
END_VAR
Upsert := THIS^.Insert_Generic(Key, Value, TRUE, bSuccess => bSuccess);
END_METHOD

END_FUNCTION_BLOCK

// POUs/Function Blocks/Collections/FB_Tree_Set
// A collection that contains no duplicate items implemented using an iterative AVL Tree.
// This data structure was implemented with the help of Max Goren's iterative AVL tree in C++. See Function Block's body for more details.
{attribute 'enable_dynamic_creation'}
{attribute 'no_assign'}
{attribute 'no_explicit_call' := 'direct call for this function block is not allowed'}
FUNCTION_BLOCK FINAL FB_Tree_Set EXTENDS FB_Collection IMPLEMENTS I_Tree_Set //, I_Enumerable, I_Copyable
VAR
	pRoot : POINTER TO T_AVL_Node;
	Traversal : T_BST_Traversal := T_BST_Traversal.In_Order; 
	pValues : POINTER TO FB_Array_List;
END_VAR

(*
	https://github.com/maxgoren
	http://www.maxgcoding.com/iterative-avl-trees-insertion/
	http://www.maxgcoding.com/iterative-avl-trees-deletion/

	MIT License
	
	Copyright (c) 2023 Max Goren
	
	Permission is hereby granted, free of charge, to any person obtaining a copy
	of this software and associated documentation files (the "Software"), to deal
	in the Software without restriction, including without limitation the rights
	to use, copy, modify, merge, publish, distribute, sublicense, and/or sell
	copies of the Software, and to permit persons to whom the Software is
	furnished to do so, subject to the following conditions:
	
	The above copyright notice and this permission notice shall be included in all
	copies or substantial portions of the Software.
	
	THE SOFTWARE IS PROVIDED "AS IS", WITHOUT WARRANTY OF ANY KIND, EXPRESS OR
	IMPLIED, INCLUDING BUT NOT LIMITED TO THE WARRANTIES OF MERCHANTABILITY,
	FITNESS FOR A PARTICULAR PURPOSE AND NONINFRINGEMENT. IN NO EVENT SHALL THE
	AUTHORS OR COPYRIGHT HOLDERS BE LIABLE FOR ANY CLAIM, DAMAGES OR OTHER
	LIABILITY, WHETHER IN AN ACTION OF CONTRACT, TORT OR OTHERWISE, ARISING FROM,
	OUT OF OR IN CONNECTION WITH THE SOFTWARE OR THE USE OR OTHER DEALINGS IN THE
	SOFTWARE.
*)

// Performs rotation and updates heights until tree is balanced.
METHOD PROTECTED Balance
VAR_INPUT
    pNode : POINTER TO T_AVL_Node;
END_VAR
VAR 
	pTmp : POINTER TO T_AVL_Node;
    Balance_Factor : T_Position;
END_VAR
WHILE pNode <> 0 AND_THEN pNode^.pParent <> 0 DO
	pTmp := pNode^.pParent;
	
	THIS^.Update_Height(pTmp);
	
	IF THIS^.Get_Balance(pTmp) < -1 THEN
		IF THIS^.Get_Balance(pTmp^.pRight) > 0 THEN THIS^.Rotate_Right(pTmp^.pRight); END_IF
		THIS^.Rotate_Left(pTmp);
		
	ELSIF THIS^.Get_Balance(pTmp) > 1 THEN
		IF THIS^.Get_Balance(pTmp^.pLeft) < 0 THEN THIS^.Rotate_Left(pTmp^.pLeft); END_IF
		THIS^.Rotate_Right(pTmp);
		END_IF
	
	pNode := pNode^.pParent;
	END_WHILE
END_METHOD

// Deletes the node and its tree/sub-trees.
{warning disable C0394}
METHOD PROTECTED Clear_Node
VAR_INPUT
	pRoot : POINTER TO T_AVL_Node;
END_VAR
VAR
	fbNode_Stack : FB_Stack;
	pTmp : POINTER TO T_AVL_Node;
END_VAR
IF pRoot = 0 THEN RETURN; END_IF

fbNode_Stack.Push(pRoot);

WHILE NOT fbNode_Stack._Empty DO
	fbNode_Stack.Get(pTmp);
	fbNode_Stack.Pop();
	
	IF pTmp^.pRight <> 0 THEN fbNode_Stack.Push(pTmp^.pRight); END_IF
	IF pTmp^.pLeft <> 0 THEN fbNode_Stack.Push(pTmp^.pLeft); END_IF
	
	THIS^.Delete_Node(pTmp);
	END_WHILE
END_METHOD

// Creates a new node in dynamic memory with a clone of the generic item as it data.
METHOD PROTECTED Create_Node : POINTER TO ST_AVL_NODE
VAR_INPUT
	Item : T_Generic;
END_VAR
Create_Node := __NEW(ST_AVL_NODE);
Create_Node^.Data := F_Clone_Generic(Item);
END_METHOD

// Safety deletes node.
// If the node and/or it's value/data is in dynamic memory it/they will be deleted.
METHOD PROTECTED Delete_Node
VAR_INPUT
	pNode : REFERENCE TO POINTER TO T_AVL_Node;
END_VAR
IF (pNode = 0) THEN RETURN; END_IF 

F_Delete_Generic(pNode^.Data);

CASE Tc2_System.F_CheckMemoryArea(pNode, 1) OF
	Tc2_System.E_TcMemoryArea.Dynamic: __DELETE(pNode);
ELSE
	pNode := 0;
	END_CASE
END_METHOD

// Finds the node with the smallest item in a tree or sub-tree.
METHOD PROTECTED Find_Minimum_Node : POINTER TO T_AVL_Node
VAR_INPUT
	pNode : POINTER TO T_AVL_Node;
END_VAR
IF pNode = 0 THEN RETURN; END_IF

WHILE pNode^.pLeft <> 0 DO
	pNode := pNode^.pLeft;
	END_WHILE
	
Find_Minimum_Node := pNode;
END_METHOD

// Gets the difference between the left and right sub-trees.
METHOD PROTECTED Get_Balance : T_Position
VAR_INPUT
	pNode : POINTER TO T_AVL_Node;
END_VAR
Get_Balance :=  THIS^.Get_Height(pNode^.pLeft) - THIS^.Get_Height(pNode^.pRight);
END_METHOD

// Safely gets the height of a sub-tree.
METHOD PROTECTED Get_Height : T_Position
VAR_INPUT
	pNode : POINTER TO T_AVL_Node;
END_VAR
Get_Height := SEL(pNode <> 0, -1, pNode^.Height);
END_METHOD

// Moves from node at source into the position of the destination.
METHOD PROTECTED Move_Node
VAR_INPUT
	pDestination, pSource : POINTER TO T_AVL_Node;
END_VAR
IF pDestination^.pParent = 0 THEN
	THIS^.pRoot := pSource;
ELSIF pDestination = pDestination^.pParent^.pLeft THEN
	pDestination^.pParent^.pLeft := pSource;
ELSE
	pDestination^.pParent^.pRight := pSource;
	END_IF
	
IF pSource <> 0 THEN
	pSource^.pParent := pDestination^.pParent;
	END_IF
END_METHOD

// Finds and removes a node from a tree/sub-tree.
METHOD PROTECTED Remove_Node
VAR_INPUT
	pNode : POINTER TO T_AVL_Node;
END_VAR
VAR
	pTmp, pSuccessor : POINTER TO T_AVL_Node;
END_VAR
pTmp := pNode;

IF pNode^.pLeft = 0 THEN
	THIS^.Move_Node(pNode, pNode^.pRight);
ELSIF pNode^.pRight = 0 THEN 
	THIS^.Move_Node(pNode, pNode^.pLeft);
ELSE
	pSuccessor := THIS^.Find_Minimum_Node(pNode^.pRight);
	IF pSuccessor^.pParent <> pNode THEN 
		THIS^.Move_Node(pSuccessor, pSuccessor^.pRight);
		pSuccessor^.pRight := pNode^.pRight;
		pSuccessor^.pRight^.pParent := pSuccessor;
		END_IF
	THIS^.Move_Node(pNode, pSuccessor);
	pSuccessor^.pLeft := pNode^.pLeft;
	pSuccessor^.pLeft^.pParent := pSuccessor;
	END_IF

THIS^.Delete_Node(pTmp);
END_METHOD

// Rotates a tree/sub-tree left.
METHOD PROTECTED Rotate_Left
VAR_INPUT
    pX : POINTER TO T_AVL_Node;
END_VAR
VAR
    pY : POINTER TO T_AVL_Node := pX^.pRight;
END_VAR
IF pY <> 0 THEN
	pX^.pRight := pY^.pLeft;
	IF pY^.pLeft <> 0 THEN pY^.pLeft^.pParent := pX; END_IF
	pY^.pParent := pX^.pParent;
	END_IF
	
IF pX^.pParent = 0 THEN
	THIS^.pRoot := pY;
ELSIF pX = pX^.pParent^.pLeft THEN
	pX^.pParent^.pLeft := pY;
ELSE
	pX^.pParent^.pRight := pY;
	END_IF
	
IF pY <> 0 THEN pY^.pLeft := pX; END_IF
	
pX^.pParent := pY;
THIS^.Update_Height(pX);
THIS^.Update_Height(pY);
END_METHOD

// Rotates a tree/sub-tree right.
METHOD PROTECTED Rotate_Right
VAR_INPUT
    pX : POINTER TO T_AVL_Node;
END_VAR
VAR
    pY : POINTER TO T_AVL_Node := pX^.pLeft;
END_VAR
IF pY <> 0 THEN
	pX^.pLeft := pY^.pRight;
	IF pY^.pRight <> 0 THEN pY^.pRight^.pParent := pX; END_IF
	pY^.pParent := pX^.pParent;
	END_IF
	
IF pX^.pParent = 0 THEN
	THIS^.pRoot := pY;
ELSIF pX = pX^.pParent^.pLeft THEN
	pX^.pParent^.pLeft := pY;
ELSE
	pX^.pParent^.pRight := pY;
	END_IF
	
IF pY <> 0 THEN pY^.pRight := pX; END_IF
	
pX^.pParent := pY;
THIS^.Update_Height(pX);
THIS^.Update_Height(pY);
END_METHOD

// Checks if an item is in a tree/ sub-tree.
METHOD PROTECTED Search_Node : POINTER TO T_AVL_Node
VAR_INPUT
	pNode : POINTER TO T_AVL_Node;
	Item : T_Generic;
END_VAR
WHILE pNode <> 0 DO
	CASE F_Compare_Generics(Item, pNode^.Data) OF
		T_Comparison.Less	: pNode := pNode^.pLeft;
		T_Comparison.Greater: pNode := pNode^.pRight; 
		T_Comparison.Equal	: 
			Search_Node := pNode;
			RETURN;
		END_CASE
	END_WHILE
END_METHOD

METHOD PROTECTED Update_Height
VAR_INPUT
	pNode : POINTER TO T_AVL_Node;
END_VAR
pNode^.Height := 1 + MAX(THIS^.Get_Height(pNode^.pLeft), THIS^.Get_Height(pNode^.pRight));
END_METHOD

// Traversal method for retrieving values in the tree set.
PROPERTY _Traversal : T_BST_Traversal
GET
_Traversal := THIS^.Traversal;
END_GET
SET
THIS^.Traversal := _Traversal;
END_SET
END_PROPERTY

// Empties/Clears/Deletes every item in the set.
METHOD Clear : I_Set
Clear := THIS^;

THIS^.Clear_Node(THIS^.pRoot);

IF THIS^.pValues <> 0 THEN  __DELETE(THIS^.pValues); END_IF

THIS^.pRoot := 0;
THIS^._Count := 0;
END_METHOD

// Checks if item is contained in set.
METHOD Contains : BOOL
VAR_INPUT
	Item : ANY; // Item to find.
END_VAR
Contains := THIS^.Search_Node(THIS^.pRoot, Item) <> 0;
END_METHOD

{attribute 'hide'}
METHOD FB_exit : BOOL
VAR_INPUT
	bInCopyCode : BOOL; // if TRUE, the exit method is called for exiting an instance that is copied afterwards (online change).
END_VAR
// If this is an online change or this collection is empty then ignore. 
IF bInCopyCode THEN RETURN; END_IF

THIS^.Clear();
END_METHOD

// Gets an immutable list of the values in the set.
{warning disable C0394}
METHOD Get_Values : I_Immutable_List
VAR_INST
	fbImmutable_List : FB_Immutable_List;
END_VAR
VAR
	pCurrent : POINTER TO T_AVL_Node;
	fbNode_Buffer : FB_Queue;
END_VAR
IF THIS^.pValues = 0 THEN THIS^.pValues := __NEW(FB_Array_List(Initial_Capacity := 0)); END_IF
fbImmutable_List(ipList := THIS^.pValues^);
Get_Values := fbImmutable_List;

THIS^.pValues^.Clear();

IF THIS^.pRoot = 0 THEN RETURN; END_IF

fbNode_Buffer.Enqueue(THIS^.pRoot);

WHILE NOT fbNode_Buffer._Empty DO
	fbNode_Buffer.Get(pCurrent).Dequeue();
	
	CASE THIS^._Traversal OF
		T_BST_Traversal.In_Order:
			IF pCurrent^.pLeft <> 0 THEN fbNode_Buffer.Enqueue_At_Front(pCurrent^.pLeft); END_IF
			THIS^.pValues^.Insert_Generic(THIS^.pValues^._Count, pCurrent^.Data);
			IF pCurrent^.pRight <> 0 THEN fbNode_Buffer.Enqueue_At_Front(pCurrent^.pRight); END_IF
			
		T_BST_Traversal.Pre_Order:
			THIS^.pValues^.Insert_Generic(THIS^.pValues^._Count, pCurrent^.Data);
			IF pCurrent^.pLeft <> 0 THEN fbNode_Buffer.Enqueue_At_Front(pCurrent^.pLeft); END_IF
			IF pCurrent^.pRight <> 0 THEN fbNode_Buffer.Enqueue_At_Front(pCurrent^.pRight); END_IF
			
		T_BST_Traversal.Post_Order:
			IF pCurrent^.pLeft <> 0 THEN fbNode_Buffer.Enqueue_At_Front(pCurrent^.pLeft); END_IF
			IF pCurrent^.pRight <> 0 THEN fbNode_Buffer.Enqueue_At_Front(pCurrent^.pRight); END_IF
			THIS^.pValues^.Insert_Generic(THIS^.pValues^._Count, pCurrent^.Data);
			
		T_BST_Traversal.Level_Order:
			THIS^.pValues^.Insert_Generic(THIS^.pValues^._Count, pCurrent^.Data);
			IF pCurrent^.pLeft <> 0 THEN fbNode_Buffer.Enqueue(pCurrent^.pLeft); END_IF
			IF pCurrent^.pRight <> 0 THEN fbNode_Buffer.Enqueue(pCurrent^.pRight); END_IF
	ELSE
		RETURN;
		END_CASE
	END_WHILE
END_METHOD

// Insert item into set.
METHOD Insert 	: I_Set
VAR_INPUT
	Item : ANY; // Data to insert
END_VAR
VAR_OUTPUT
	bSuccess : BOOL; // Indicates whether operation was successful. Success = TRUE, Failure = FALSE
END_VAR
Insert := THIS^.Insert_Generic(Item, bSuccess => bSuccess);
END_METHOD

// Adds new generic item at into set.
// The set will store a copy of the generic item so as to not modify the original value outside it's scope.
METHOD Insert_Generic : I_Set
VAR_INPUT
	Item : T_Generic; // Item to store
END_VAR
VAR_OUTPUT
	bSuccess : BOOL; // Indicates whether operation was successful. Success = TRUE, Failure = FALSE
END_VAR
VAR
	pCurrent, pPrevious : POINTER TO T_AVL_Node;
END_VAR
Insert_Generic := THIS^;

pCurrent := THIS^.pRoot;
pPrevious := pCurrent;

WHILE pCurrent <> 0 DO
	pPrevious := pCurrent;
	CASE F_Compare_Generics(Item, pCurrent^.Data) OF
		T_Comparison.Less 	 : pCurrent := pCurrent^.pLeft;
		T_Comparison.Greater : pCurrent := pCurrent^.pRight;
		T_Comparison.Equal 	 : RETURN;
	ELSE
		THIS^._Error_Status := F_Error(TRUE, GVL_Errors.ERR_NOT_SUPPORTED, 'Invalid comparison.');
		RETURN;
		END_CASE
	END_WHILE

pCurrent := THIS^.Create_Node(Item);

IF pPrevious = 0 THEN
	THIS^.pRoot := pCurrent;
ELSE
	CASE F_Compare_Generics(Item, pPrevious^.Data) OF
		T_Comparison.Less: pPrevious^.pLeft := pCurrent;
	ELSE
		pPrevious^.pRight := pCurrent;
		END_CASE
	END_IF

pCurrent^.pParent := pPrevious;
	
THIS^.Balance(pCurrent);

bSuccess := TRUE;
THIS^.Increment_Count();
THIS^.Clear_Error();
END_METHOD

// Removes item from the set.
METHOD Remove : I_Set
VAR_INPUT
	Item : ANY; // Data to remove
END_VAR
VAR_OUTPUT
	bSuccess : BOOL; // Indicates whether operation was successful. Success = TRUE, Failure = FALSE
END_VAR
Remove := THIS^.Remove_Generic(Item, bSuccess => bSuccess);
END_METHOD

// Removes generic item from the set.
METHOD Remove_Generic : I_Set
VAR_INPUT
	Item : T_Generic; // Data to remove
END_VAR
VAR_OUTPUT
	bSuccess : BOOL; // Indicates whether operation was successful. Success = TRUE, Failure = FALSE
END_VAR
VAR
	pTmp : POINTER TO T_AVL_Node;
END_VAR
Remove_Generic := THIS^;

pTmp := THIS^.Search_Node(THIS^.pRoot, Item);

IF pTmp = 0 THEN RETURN; END_IF

THIS^.Remove_Node(pTmp);
THIS^.Balance(pTmp);

bSuccess := TRUE;
THIS^.Decrement_Count();
THIS^.Clear_Error();

IF THIS^._Empty THEN THIS^.pRoot := 0; END_IF
END_METHOD

END_FUNCTION_BLOCK

// POUs/Function Blocks/Enumerators/FB_Enumerator
// Base function block for enumerators.
{attribute 'enable_dynamic_creation'}
{attribute 'no_explicit_call' := 'direct call for this function block is not allowed'}
FUNCTION_BLOCK ABSTRACT FB_Enumerator IMPLEMENTS I_Enumerator
VAR
	ipEnumerator : REFERENCE TO I_Enumerator;
	Index : T_Position := -1;
END_VAR

// Gets an item in the collection at current positon of the enumerator.
METHOD ABSTRACT Current : I_Enumerator
VAR_INPUT
	Item : ANY;
END_VAR
END_METHOD

// Gets an item in the collection at current positon of the enumerator as a string.
METHOD ABSTRACT Current_As_String : I_Enumerable
VAR_INPUT
	sItem : REFERENCE TO STRING;
END_VAR
END_METHOD

// Releases resources allocated to the enumerator. Returns TRUE if successful.
METHOD FINAL Dispose : BOOL
IF __ISVALIDREF(THIS^.ipEnumerator) THEN RETURN; END_IF
THIS^.ipEnumerator := 0;
__DELETE(THIS);
END_METHOD

{attribute 'hide'}
METHOD ABSTRACT FB_exit : BOOL
VAR_INPUT
	bInCopyCode : BOOL; // if TRUE, the exit method is called for exiting an instance that is copied afterwards (online change).
END_VAR
END_METHOD

{attribute 'hide'}
METHOD FB_init : BOOL
VAR_INPUT
	bInitRetains : BOOL; // if TRUE, the retain variables are initialized (warm start / cold start)
	bInCopyCode : BOOL;  // if TRUE, the instance afterwards gets moved into the copy code (online change)
	ipEnumerator : REFERENCE TO I_Enumerator;
END_VAR
IF bInCopyCode OR_ELSE NOT __ISVALIDREF(ipEnumerator) THEN RETURN; END_IF
IF ipEnumerator <> 0 THEN ipEnumerator.Dispose(); END_IF
THIS^.ipEnumerator REF= ipEnumerator;
END_METHOD

// Advances the enumerator to the next item of the collection.
METHOD ABSTRACT Next : BOOL
END_METHOD

// Sets the enumerator to its initial position, which is before the first element in the collection.
METHOD ABSTRACT Reset : I_Enumerator
END_METHOD

END_FUNCTION_BLOCK

// POUs/Function Blocks/Misc/FB_Free
// Frees pointer when this instance of the FB leaves the scope;
{attribute 'no_explicit_call' := 'direct call for this function block is not allowed'}
FUNCTION_BLOCK INTERNAL FINAL FB_Free
VAR
	_pValue : REFERENCE TO POINTER TO BYTE;
END_VAR

{attribute 'hide'} 
METHOD FB_exit : BOOL
VAR_INPUT
	bInCopyCode : BOOL; // if TRUE, the exit method is called for exiting an instance that is copied afterwards (online change).
END_VAR
IF bInCopyCode THEN RETURN; END_IF
IF NOT __ISVALIDREF(THIS^._pValue) THEN RETURN; END_IF
IF THIS^._pValue <> 0 THEN __DELETE(THIS^._pValue); END_IF
END_METHOD

{attribute 'hide'} 
{attribute 'no_explicit_call' := 'do not call this POU directly'}
METHOD FB_init : BOOL
VAR_INPUT
	bInitRetains 	: BOOL; // if TRUE, the retain variables are initialized (warm start / cold start)
	bInCopyCode 	: BOOL;  // if TRUE, the instance afterwards gets moved into the copy code (online change)
	pValue 			: REFERENCE TO POINTER TO BYTE; // Pointer to be freed on exit
END_VAR
THIS^._pValue REF= pValue;
END_METHOD

END_FUNCTION_BLOCK

// POUs/Functions/F_Any_To_Generic
FUNCTION F_Any_To_Generic : T_Generic
VAR_INPUT
	Value : ANY;
END_VAR

F_Any_To_Generic := Value;

END_FUNCTION

// POUs/Functions/F_Compare_Any
// Compares value A to generic value B of any type and returns the evaluation.
FUNCTION F_Compare_Any : T_Comparison
VAR_INPUT
	A : ANY;
	B : ANY;
END_VAR

F_Compare_Any := F_Compare_Generics(A, B);

END_FUNCTION

// POUs/Functions/F_String_To_Any
// Converts string to generic, returns TRUE if successful.
FUNCTION F_String_To_Any : BOOL
VAR_INPUT
	sValue : REFERENCE TO STRING;
	Value : ANY;
END_VAR
VAR
	pBool			: POINTER TO BOOL;
    pByte			: POINTER TO BYTE;
    pWord			: POINTER TO WORD;
    pDWord			: POINTER TO DWORD;
    pLWord			: POINTER TO LWORD;
    pSint			: POINTER TO SINT;
    pInt			: POINTER TO INT;
    pDint			: POINTER TO DINT;
    pLint			: POINTER TO LINT;
    pUSint			: POINTER TO USINT;
    pUInt			: POINTER TO UINT;
    pUDint			: POINTER TO UDINT;
    pULint			: POINTER TO ULINT;
    pReal			: POINTER TO REAL;
    pLReal			: POINTER TO LREAL;
    pString			: POINTER TO STRING(255);
    pWString		: POINTER TO WSTRING;
    pTime			: POINTER TO TIME;
    pDate			: POINTER TO DATE;
    pDate_And_Time	: POINTER TO DATE_AND_TIME;
    pTime_Of_Day	: POINTER TO TIME_OF_DAY;
    pPointer		: POINTER TO PVOID;
	pLTime 			: POINTER TO LTIME;
END_VAR

IF (Value.pValue = 0) OR_ELSE (NOT F_String_Convertable_Generic(Value)) OR_ELSE (NOT __ISVALIDREF(sValue)) THEN RETURN; END_IF;

F_String_To_Any := TRUE;

CASE Value.TypeClass OF 
	__SYSTEM.TYPE_CLASS.TYPE_BOOL:
		pBool := Value.pValue;
		pBool^ := TO_BOOL(sValue);
		
    __SYSTEM.TYPE_CLASS.TYPE_BYTE:
		pByte := Value.pValue;
		pByte^ := TO_BYTE(sValue);
		
    __SYSTEM.TYPE_CLASS.TYPE_WORD:
		pWord := Value.pValue;
		pWord^ := TO_WORD(sValue);
		
    __SYSTEM.TYPE_CLASS.TYPE_DWORD:
		pDWord := Value.pValue;
		pDWord^ := TO_DWORD(sValue);
		
    __SYSTEM.TYPE_CLASS.TYPE_LWORD:
		pLWord := Value.pValue;
		pLWord^ := TO_LWORD(sValue);
		
    __SYSTEM.TYPE_CLASS.TYPE_SINT:
		pSint := Value.pValue;
		pSint^ := TO_SINT(sValue);
		
    __SYSTEM.TYPE_CLASS.TYPE_INT:
		pInt := Value.pValue;
		pInt^ := TO_INT(sValue);
		
    __SYSTEM.TYPE_CLASS.TYPE_DINT:
		pDint := Value.pValue;
		pDint^ := TO_DINT(sValue);
		
    __SYSTEM.TYPE_CLASS.TYPE_LINT:
		pLint := Value.pValue;
		pLint^ := TO_LINT(sValue);
		
    __SYSTEM.TYPE_CLASS.TYPE_USINT:
		pUSint := Value.pValue;
		pUSint^ := TO_USINT(sValue);
		
    __SYSTEM.TYPE_CLASS.TYPE_UINT:
		pUInt := Value.pValue;
		pUInt^ := TO_UINT(sValue);
		
    __SYSTEM.TYPE_CLASS.TYPE_UDINT:
		pUDint := Value.pValue;
		pUDint^ := TO_UDINT(sValue);
		
    __SYSTEM.TYPE_CLASS.TYPE_ULINT:
		pULint := Value.pValue;
		pULint^ := TO_ULINT(sValue);
		
   __SYSTEM.TYPE_CLASS.TYPE_REAL:
		pReal := Value.pValue;
		pReal^ := TO_REAL(sValue);
		
    __SYSTEM.TYPE_CLASS.TYPE_LREAL:
		pLReal := Value.pValue;
		pLReal^ := TO_LREAL(sValue);
		
    __SYSTEM.TYPE_CLASS.TYPE_STRING:
		Tc2_Utilities.STRNCPY(Value.pValue, ADR(sValue), Value.diSize); 
		
   __SYSTEM.TYPE_CLASS.TYPE_WSTRING:
   		Tc2_Utilities.STRING_TO_WSTRING2(Value.pValue, ADR(sValue), TO_UDINT(Value.diSize));
		
    __SYSTEM.TYPE_CLASS.TYPE_TIME:
		pTime := Value.pValue;
		pTime^ := TO_TIME(sValue);
		
	__SYSTEM.TYPE_CLASS.TYPE_LTIME:
		pLTime := Value.pValue;
		pLTime^ := TO_LTIME(sValue);
		
    __SYSTEM.TYPE_CLASS.TYPE_DATE:
		pDate := Value.pValue;
		pDate^ := TO_DATE(sValue);
		
    __SYSTEM.TYPE_CLASS.TYPE_DATEANDTIME:
		pDate_And_Time := Value.pValue;
		pDate_And_Time^ := TO_DT(sValue);
		
    __SYSTEM.TYPE_CLASS.TYPE_TIMEOFDAY:
		pTime_Of_Day := Value.pValue;
		pTime_Of_Day^ := TO_TOD(sValue);
	
	__SYSTEM.TYPE_CLASS.TYPE_POINTER:
		pPointer := Value.pValue;
		pPointer^ := Tc2_Utilities.STRING_TO_PVOID(sValue);
END_CASE

END_FUNCTION

// POUs/MAIN
PROGRAM INTERNAL MAIN
VAR
	i,j : T_Position;
	Comp : T_Comparison;
	bAdd, bRemove, bClear : BOOL;
	fbArray : FB_Array(10);
	fbArray_List : FB_Array_List(0);
	fbList : FB_List;
	fbQueue : FB_Queue;
	fbSet : FB_Tree_Set;
	fbMap : FB_Tree_Map;
	fbDeque : FB_Deque;
	Data : ARRAY[0..10] OF INT := [1,2,3,4,5,6,7,8,9,10];
END_VAR

Comp := F_Compare_Any(i,j);

IF bAdd THEN
	bAdd := FALSE;
	fbQueue
		.Enqueue(Data[0])
		.Enqueue(Data[1])
		.Reverse();
	END_IF

IF bRemove THEN 
	bRemove := FALSE;
	fbSet.Remove(j);
	END_IF
	
IF bClear THEN 
	bClear := FALSE;
	fbSet.Clear();
	END_IF

END_PROGRAM

// Project Information/F_GetCompany
// This function has been automatically generated from the project information.
{attribute 'signature_flag' := '1073741824'}
{attribute 'TcGenerated'}
{attribute 'no-analysis'}
FUNCTION F_GetCompany : WSTRING
VAR_INPUT
	
END_VAR

F_GetCompany := "FisoThemes";

END_FUNCTION

// Project Information/F_GetTitle
// This function has been automatically generated from the project information.
{attribute 'signature_flag' := '1073741824'}
{attribute 'TcGenerated'}
{attribute 'no-analysis'}
FUNCTION F_GetTitle : WSTRING
VAR_INPUT
	
END_VAR

F_GetTitle := "TwinCat Dynamic Collections";

END_FUNCTION

// Project Information/F_GetVersion
// This function has been automatically generated from the project information.
{attribute 'signature_flag' := '1073741824'}
{attribute 'TcGenerated'}
{attribute 'no-analysis'}
FUNCTION F_GetVersion : ST_LibVersion
VAR_INPUT
	
END_VAR

F_GetVersion.iMajor := 1;
F_GetVersion.iMinor := 0;
F_GetVersion.iBuild := 1;
F_GetVersion.iRevision := 7;

END_FUNCTION
